TYPE "Positioning_DOL_Machine_Alr"
VERSION : 0.1
// Block: Positioning_DOL_Machine_Alr
   STRUCT
      Ax : OOAx_Alr;
      Ax_NotHomed : Bool;
      S120 : Struct
         Drive : Bool;
      END_STRUCT;
      S120_ComErr : Bool;
      BrakeTimeOut : Bool;
      Fan_M : MotorAlr;
   END_STRUCT;

END_TYPE
